DATA_BLOCK "ST10_SystemModeFB_iDB"
{ S7_Optimized_Access := 'TRUE' }
VERSION : 0.1
NON_RETAIN
"SystemMode"

BEGIN

END_DATA_BLOCK

